// TIA Portal V17 export
FUNCTION_BLOCK "ConveyorControl"   // FB500, LAD
AUTHOR : Giacomo P.
FAMILY : SPIN_SRL
// stored: SetENOAutomatically true, UDABlockProperties GENERATED_BY_XMLREADER, UDAEnableTagReadback true
   VAR_INPUT
      iSensor : Bool;
      iRun : Bool;
   END_VAR
   VAR_OUTPUT
      oConveyor : Bool;
   END_VAR
BEGIN

REGION Network 1: 传送带控制
   // Run=1 且 Sensor=0 时 Conveyor=1；Sensor=1 或 Run=0 时 Conveyor=0
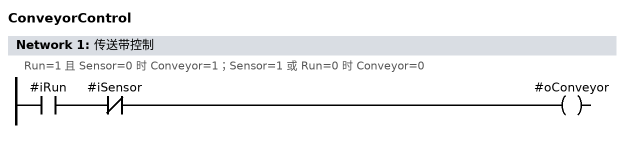
   RUNG wire#powerrail
      Contact( #iRun )
      I_Contact( #iSensor )
      Coil( #oConveyor )
   END_RUNG
   // the same network as SCL:
   #oConveyor := #iRun AND NOT #iSensor;
END_REGION
END_FUNCTION_BLOCK
